// TwinCAT 3 PLC project Untitled1
// ProgramVersion: 3.1.4024.0
// libraries:
//   Tc2_Standard, * (Beckhoff Automation GmbH)
//   Tc2_System, * (Beckhoff Automation GmbH)
//   Tc2_Utilities, * (Beckhoff Automation GmbH)
//   Tc3_Module, * (Beckhoff Automation GmbH)
//   VisuDialogs, * (System)
//   VisuSymbols,3.5.10.0,System
// project tree:
//   / Class Diagram.TcCD (not stored), GlobalTextList.TcGTLO, PlcTask.TcTTO, Visualization Manager.TcVMO (not stored)
//   GVLs/ gCONSTANT.TcGVL
//   LampUnit/ E_Command.TcDUT, FB_Button.TcPOU, FB_Unit.TcPOU
//   Logger/ FB_Logger.TcPOU, I_Log.TcIO
//   POUs/ MAIN.TcPOU
//   VISUs/ Visualization.TcVIS, UserControlButton.TcVIS
// real-time tasks:
//   TASK PlcTask: cycle T#70000us, priority 20, ADS port 350

CONFIGURATION Untitled1
    RESOURCE PLC ON TwinCAT3
        TASK PlcTask(INTERVAL := T#10ms, PRIORITY := 20);
        PROGRAM MAIN WITH PlcTask : MAIN;
    END_RESOURCE
END_CONFIGURATION

// ---- LampUnit/E_Command.TcDUT
{attribute 'qualified_only'}
{attribute 'strict'}
{attribute 'to_string'}
TYPE E_Command :
(
	Forward := 0,
	Stop := 1,
	Backward := 2,
	Generate := 3
);
END_TYPE

// ---- GVLs/gCONSTANT.TcGVL
//{attribute 'qualified_only'}
VAR_GLOBAL CONSTANT
	MAX_UNIT_NUMBER : BYTE := 9;
//	MIN_UNIT_NUMBER_STRING : STRING := '1';
//	MAX_UNIT_NUMBER_STRING : STRING := BYTE_TO_STRING(MAX_UNIT_NUMBER);
END_VAR

// ---- Logger/I_Log.TcIO
INTERFACE I_Log

METHOD AddLog : BOOL
VAR_INPUT
	sLog : STRING;
END_VAR
END_METHOD

END_INTERFACE

// ---- POUs/MAIN.TcPOU
PROGRAM MAIN
VAR
	fbUnit : FB_Unit;
	fbLogger : FB_Logger;
END_VAR

fbUnit.Initalize(fbLogger);
fbUnit();

fbLogger.Write('C:/Test.csv');

END_PROGRAM

// ---- LampUnit/FB_Unit.TcPOU
FUNCTION_BLOCK FB_Unit
VAR
	step : (idle, init, Forward, Backward, Stop);
	Command : E_Command;
	fbTon : TON := (PT:=T#1S);
	bInit : BOOL;
	i : INT;
	
	
	(*Visu*)
	LED : ARRAY[1..10] OF BOOL;
	LEDLocation : ARRAY[1..2] OF INT;
	
	GenerateButton : FB_Button(E_Command.Generate);
	ForwardButton : FB_Button(E_Command.Forward);
	BackwardButton : FB_Button(E_Command.Backward);
	StopButton : FB_Button(E_Command.Stop);
END_VAR

IF NOT bInit THEN
	RETURN;
END_IF

IF Command = E_Command.Generate THEN
	LEDLocation[1] := 1;
	LEDLocation[2] := 2;
	step := Init;
	fbTon(IN := FALSE);
END_IF

CASE step OF
	Idle:
		;
	init:		
		fbTon(IN := TRUE);
		IF fbTon.Q THEN
			fbTon(IN := FALSE);
			IF Command = E_Command.Forward THEN
				step := Forward;
			ELSIF Command = E_Command.Backward THEN
				step := Backward;
			ELSIF Command = E_Command.Stop THEN
				step := Stop;
				fbTon(IN := FALSE);
			END_IF
		END_IF
	Forward:
		FOR i:= 1 TO 2 BY 1 DO
			IF LEDLocation[i] > 0 AND LEDLocation[i] <= 10 THEN
				LEDLocation[i] := LEDLocation[i] + 1;
			ELSE
				LEDLocation[i] := 0;
			END_IF 
		END_FOR
		fbTon(IN := TRUE);
		step := Init;
		
	Backward:
		FOR i:= 1 TO 2 BY 1 DO
			IF LEDLocation[i] > 0 AND LEDLocation[i] < 11 THEN
				LEDLocation[i] := LEDLocation[i] - 1;
			ELSE
				LEDLocation[i] := 0;
			END_IF 
		END_FOR
		fbTon(IN := TRUE);
		step := Init;
		
	Stop:
		IF Command = E_Command.Forward THEN
			fbTon(IN := TRUE);
			IF fbTon.Q THEN
				step := Forward;
				fbTon(IN := FALSE);
			END_IF
		ELSIF Command = E_Command.Backward THEN
			fbTon(IN := TRUE);
			IF fbTon.Q THEN
				step := Backward;
				fbTon(IN := FALSE);
			END_IF
		END_IF
END_CASE

TurnOnTwoLED(LEDLocation[1],LEDLocation[2]);
ForwardButton();
BackwardButton();
StopButton();
GenerateButton();

METHOD Initalize : BOOL
VAR_INPUT
	iLog : I_Log;
END_VAR
IF bInit THEN
	RETURN;
END_IF
ForwardButton.iLog := iLog;
ForwardButton.refCommand REF= Command;
BackwardButton.iLog := iLog;
BackwardButton.refCommand REF= Command;
StopButton.iLog := iLog;
StopButton.refCommand REF= Command;
GenerateButton.iLog := iLog;
GenerateButton.refCommand REF= Command;

bInit := TRUE;
END_METHOD

METHOD PRIVATE TurnOnTwoLED
VAR_INPUT
	Location1 : INT;
	Location2 : INT;
END_VAR
VAR
	i : INT;
END_VAR
IF Location1 = 0 AND Location2 = 0 THEN
	step := Idle;
END_IF

FOR i := 1 TO 10 BY 1 DO
	IF i = Location1 THEN
		LED[i] := TRUE;
	ELSIF i = Location2 THEN
		LED[i] := TRUE;
	ELSE
		LED[i] := FALSE;
	END_IF
END_FOR
END_METHOD

END_FUNCTION_BLOCK

// ---- LampUnit/FB_Button.TcPOU
FUNCTION_BLOCK FB_Button
VAR
	sButtonName : STRING;
	bExecute : BOOL;
	ExecuteCounter : UDINT;
	_refCommand : REFERENCE TO E_Command;
	InputCommand : E_Command;
	_iLog : I_Log;
	Rtrig : R_TRIG;
END_VAR

IF bExecute THEN
	ExecuteCounter := ExecuteCounter + _TaskInfo[1].CycleTime/10000;
	IF ExecuteCounter >= 1000 THEN
		_refCommand := InputCommand;
		bExecute := FALSE;
	END_IF
ELSE
	ExecuteCounter := 0;
END_IF

Rtrig(CLK := bExecute);
IF Rtrig.Q THEN
	_iLog.AddLog(CONCAT(TO_STRING(InputCommand),' is pushed'));
END_IF

METHOD FB_init : BOOL
VAR_INPUT
	bInitRetains : BOOL; // if TRUE, the retain variables are initialized (warm start / cold start)
	bInCopyCode : BOOL;  // if TRUE, the instance afterwards gets moved into the copy code (online change)
	InputCommand : E_Command;
END_VAR
sButtonName := TO_STRING(InputCommand);
THIS^.InputCommand := InputCommand;
END_METHOD

PROPERTY iLog : I_Log
GET
iLog := _iLog;
END_GET
SET
_iLog := iLog;
END_SET
END_PROPERTY

PROPERTY refCommand : REFERENCE TO E_COMMAND
GET
refCommand REF= _refCommand;
END_GET
SET
 _refCommand REF= refCommand;
END_SET
END_PROPERTY

END_FUNCTION_BLOCK

// ---- Logger/FB_Logger.TcPOU
FUNCTION_BLOCK FB_Logger IMPLEMENTS I_Log
VAR
	arrLog : ARRAY[1..MAX_LOG_INDEX] OF STRING;
	fbLocalTime : FB_LocalSystemTime;
	sCurrentTime : STRING;
	fbRingBuffer : FB_MemRingBuffer;
	buffer : ARRAY[1..1000] OF BYTE;
	
	fbFileWrite : FB_FileWrite;
	fbFileOpen : FB_FileOpen;
	fbFileClose : FB_FileClose;
END_VAR

METHOD AddLog : BOOL
VAR_INPUT
	sLog : STRING;
END_VAR
VAR
	i:INT;
END_VAR
fbLocalTime(bEnable := TRUE);
sCurrentTime := SYSTEMTIME_TO_STRING(fbLocalTime.systemTime);
IF arrLog[10] <> '' THEN
	fbRingBuffer.A_AddTail(pWrite := ADR(arrLog[10]), cbWrite := INT_TO_UDINT(LEN(arrLog[10])+1), pBuffer := ADR(Buffer), cbBuffer := SIZEOF(Buffer));
END_IF

FOR i := MAX_LOG_INDEX TO 2 BY -1 DO
	arrLog[i] := arrLog[i-1];
END_FOR
arrLog[1] := CONCAT(sCurrentTime, ': ');
arrLog[1] := CONCAT(arrLog[1], sLog);
END_METHOD

METHOD Write : BOOL;
VAR_INPUT
	sPath : T_MaxString;
END_VAR
VAR_INST
	step : INT;
	sString : STRING;
	arrTest : ARRAY[1..100] OF BYTE;
END_VAR
fbLocalTime(bEnable := TRUE);
CASE step OF
	0:
		fbFileOpen(bExecute := FALSE);
		fbFileWrite(bExecute := FALSE);
		fbFileClose(bExecute := FALSE);
		fbRingBuffer.A_RemoveHead(pRead := ADR(sString), cbRead := SIZEOF(sString));
		IF fbRingBuffer.bOk THEN
			step := 10;
			sString := CONCAT(sString,',$N');
			MEMSET(ADR(arrTest),0,SIZEOF(arrTest));
			MEMCPY(ADR(arrTest),ADR(sString),INT_TO_UDINT(LEN(sString)));
		END_IF
	10:
	
	fbFileOpen(
		sNetId:= , 
		sPathName:= sPath, 
		nMode:= FOPEN_MODEAPPEND OR FOPEN_MODETEXT, 
		bExecute:= TRUE, 
		hFile=> );
	IF NOT fbFileOpen.bBusy THEN
		step := 20;
	END_IF
		
	20:
	fbFileWrite(
		sNetId:= , 
		hFile:= fbFileOpen.hFile, 
		pWriteBuff:= ADR(sString), 
		cbWriteLen:= INT_TO_UDINT(LEN(sString)), 
		bExecute:= TRUE, 
		);
	IF NOT fbFileWrite.bBusy THEN
		IF fbRingBuffer.nCount >= 1 THEN
			step := 0;
		ELSE
			step := 30;
		END_IF
	END_IF
	
	30:
	fbFileClose(
		sNetId:= , 
		hFile:= fbFileOpen.hFile, 
		bExecute:= TRUE, 
		tTimeout:= , 
		bBusy=> , 
		bError=> , 
		nErrId=> );
	IF NOT fbFileClose.bBusy THEN
		step := 0;
		Write := TRUE;
	END_IF
END_CASE
END_METHOD

END_FUNCTION_BLOCK

// ---- GlobalTextList.TcGTLO
TEXTLIST GlobalTextList
  809 = '%n'
  480 = '%s'
  795 = '1'
  146 = 'Log'
  599 = 'Receive Able'
  297 = 'Receive Complete'
  69 = 'Receive Start'
  293 = 'Send Able'
  929 = 'Send Complete'
  688 = 'Send Start'
  445 = '생성'
  184 = '실행'
  373 = '전진'
  274 = '정지'
  558 = '후진'
END_TEXTLIST

// ---- VISUs/Visualization.TcVIS
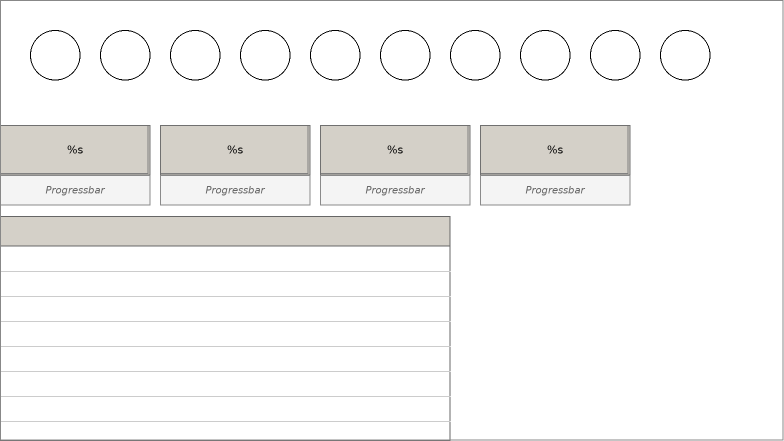
VISUALIZATION Visualization  // 784x441
    Ellipse (30,30 50x50)
        toggle MAIN.fbUnit.LED[1]
    Ellipse (100,30 50x50)
        toggle MAIN.fbUnit.LED[2]
    Ellipse (170,30 50x50)
        toggle MAIN.fbUnit.LED[3]
    Ellipse (240,30 50x50)
        toggle MAIN.fbUnit.LED[4]
    Ellipse (310,30 50x50)
        toggle MAIN.fbUnit.LED[5]
    Ellipse (380,30 50x50)
        toggle MAIN.fbUnit.LED[6]
    Ellipse (450,30 50x50)
        toggle MAIN.fbUnit.LED[7]
    Ellipse (520,30 50x50)
        toggle MAIN.fbUnit.LED[8]
    Ellipse (590,30 50x50)
        toggle MAIN.fbUnit.LED[9]
    Ellipse (660,30 50x50)
        toggle MAIN.fbUnit.LED[10]
    Polygon (783,215)
    Frame (0,125 150x80)
        shows UserControlButton(bExecute := MAIN.fbUnit.GenerateButton.bExecute, Counter := MAIN.fbUnit.GenerateButton.ExecuteCounter, sName := MAIN.fbUnit.GenerateButton.sButtonName)
    Frame (160,125 150x80)
        shows UserControlButton(bExecute := MAIN.fbUnit.ForwardButton.bExecute, Counter := MAIN.fbUnit.ForwardButton.ExecuteCounter, sName := MAIN.fbUnit.ForwardButton.sButtonName)
    Frame (320,125 150x80)
        shows UserControlButton(bExecute := MAIN.fbUnit.BackwardButton.bExecute, Counter := MAIN.fbUnit.BackwardButton.ExecuteCounter, sName := MAIN.fbUnit.BackwardButton.sButtonName)
    Frame (480,125 150x80)
        shows UserControlButton(bExecute := MAIN.fbUnit.StopButton.bExecute, Counter := MAIN.fbUnit.StopButton.ExecuteCounter, sName := MAIN.fbUnit.StopButton.sButtonName)
    Table (0,216 450x225), data array: MAIN.fbLogger.arrLog
        p3854506369: MAIN.fbLogger.arrLog[INDEX]
END_VISUALIZATION

// ---- VISUs/UserControlButton.TcVIS
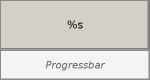
VISUALIZATION UserControlButton  // 150x80
VAR_IN_OUT
	bExecute : BOOL;
	Counter : UDINT;
	sName : STRING;
END_VAR
    Button (0,0 150x50), "%s", text variable: sName
        tap bExecute
        OnMouseDown: execute {  }
    Progressbar (0,50 150x30), variable: Counter
END_VISUALIZATION
